{attribute 'qualified_only'}
{attribute 'strict'}
TYPE BagDetectionStatus:
(
    UNKNOWN := 0,
    OKAY := 1,
    NG := 2,
	ERROR := 3
);
END_TYPE

(* stored: Version 1.1.0.1, ProductVersion 3.1.4024.12
   DUT BagDetectionStatus: Id {419dd7a7-cc3b-4aa6-ae5c-d664d1c4d4fc} *)
